PROGRAM EX_Error
VAR_IN_OUT
	Station		:structStationCtrl;
END_VAR

VAR
END_VAR

IF MC.ResetPressed THEN
	Station.SeqFaultWord := 0;
END_IF

(* 	Reserved Station.SeqFaultWord 
	= 1~49 for Major Fault
	= 100~149 for Origin Sequence Fault
	= 150~199 for Origin Width Adjust Sequence Fault
	= 200~299 for Auto Sequence Fault
	= 300~399 for misc fault listed on this page*)

Station.MajorFault := (Station.SeqFaultWord > 0) AND (Station.SeqFaultWord < 50);
Station.MinorFault := (Station.SeqFaultWord >= 100) OR 	Station.DeviceFault OR 
														E_WT_Conv_Jam OR 
														E_Weight_CV_CartonNotDetect or
														E_CartonTapingErrL OR 
														E_CartonTapingErrL;

END_PROGRAM

(* stored: Version 1.1.0.1, ProductVersion 3.1.4018.2
   POU EX_Error: Id {cd490844-37de-46d4-b5f0-5a0023795cfd}, SpecialFunc None *)
